FUNCTION_BLOCK ABSTRACT FB_Test IMPLEMENTS ITest
VAR
	_name			: STRING;
	_message		: STRING[255];
END_VAR

METHOD PROTECTED AssertEquals : BOOL
VAR_INPUT
	expected		: ANY;
	result			: ANY;
	failmsg			: STRING[255];
END_VAR
VAR
	sExp, sRes		: STRING;
END_VAR
IF (expected.diSize <> result.diSize) THEN
	_message := 'Test error: expected value type mismatch';
	AssertEquals := FALSE;
	RETURN;
END_IF

IF (Expected.pValue^ <> Result.pValue^) THEN
	sExp := CONCAT(' Expected: ', TO_STRING(expected.pValue^));
	sRes := CONCAT(' Result: ', TO_STRING(result.pValue^));
	_message := CONCAT(CONCAT(failmsg, sExp), sRes);
	AssertEquals := FALSE;
ELSE
	AssertEquals := TRUE;
END_IF
END_METHOD

{attribute 'TcRpcEnable'}
METHOD Execute : BOOL
VAR
END_VAR
END_METHOD

METHOD FB_init : BOOL
VAR_INPUT
	bInitRetains : BOOL; // if TRUE, the retain variables are initialized (warm start / cold start)
	bInCopyCode : BOOL;  // if TRUE, the instance afterwards gets moved into the copy code (online change)
	sName : STRING;
END_VAR
_name := sName;
END_METHOD

{attribute ‘monitoring’ := ‘call’}
PROPERTY PUBLIC Message : STRING(255)
GET
Message := _message;
END_GET
END_PROPERTY

{attribute ‘monitoring’ := ‘call’}
PROPERTY PUBLIC Name : STRING
GET
Name := _name;
END_GET
END_PROPERTY

END_FUNCTION_BLOCK

(* stored: Version 1.1.0.1, ProductVersion 3.1.4024.12
   POU FB_Test: Id {8831bd5e-bd34-44b6-83a6-6d659c4588f7}, SpecialFunc None
   Method AssertEquals: Id {b7f9f968-56cb-477a-b18f-fd7d7ae6de0b}
   Method Execute: Id {935cc836-92fd-4164-acc4-799697454b33}
   Method FB_init: Id {5da565e2-8a36-4cb2-a7c8-234d759f9b2c}
   Property Message: Id {a709b7be-4f75-4801-b015-50eb314430df}
   Get Get: Id {5c414332-42b2-45f0-85a8-b658be172896}
   Property Name: Id {b5b974e6-5d92-4d7e-965e-971dd3c7cf74}
   Get Get: Id {f6d5d1b3-9f88-44e2-a9e2-69032c9fc677} *)
